{region '#Template'}
	{attribute 'Version' := '6.0.3.0'}
	{attribute 'Tags' := '"LCID": "1031", "Text": "AC, Allgemein, AHU, Startprogramm, Aggregat, Kommandierung"'}
	{attribute 'Tags' := '"LCID": "1033", "Text": "AC, General, AHU, Start program, Aggregate, Command"'}
	{attribute 'Using' := '"Type": "Template", "URI": "E_BA_AC_PlantStep01"'}
	{attribute 'Using' := '"Type": "Template", "URI": "E_BA_AC_OpMod01"'}
	{attribute 'Using' := '"Type": "Template", "URI": "Priority"'}
	{attribute 'Description' := '"LCID": "1031", "Text": "Kommandierung der Anlage FB_BA_AHU_1st_10"'}
	{attribute 'Description' := '"LCID": "1033", "Text": "Commanding the plant FB_BA_AHU_1st_10"'}
{endregion}

FUNCTION_BLOCK FB_BA_AC_PlantCmd_AHU_1st_10 EXTENDS FB_BA_View
VAR_INPUT
	eOpMode						: E_BA_AC_OpMod01;
END_VAR
VAR_OUTPUT
	ePltStp						: E_BA_AC_PlantStep01;	//	Stufen des Anlagenstarts	//	Stages of the plant starts	
	bStepCtrlUp					: BOOL;
	bStepCtrlDown				: BOOL;	
END_VAR
VAR_IN_OUT
	arrAggregate				: ARRAY [1..MAX(1,BA_Param.nMaxAggregate)] OF ST_BA_Aggregate;
END_VAR
VAR_INPUT CONSTANT
	DmpDlyCls					: FB_BA_AV_Op;
	SuAFanDlyOn					: FB_BA_AV_Op;
	ExtAFanDlyOn				: FB_BA_AV_Op;
	TempCtrlDlyOn				: FB_BA_AV_Op;
	PltStp						: FB_BA_MV_Op;
	PlantControl				: FB_BA_PlantControl;
END_VAR
VAR_INPUT CONSTANT PERSISTENT
	bInit						: BOOL := TRUE;
END_VAR
VAR
	MMuxStart					: FB_BA_MMUX_B16;
	MMuxProfile					: FB_BA_MMUX_UDI16;
	MMuxPltStp					: FB_BA_MMUX_UDI16;	//	Stufen des Anlagenstarts	//	Stages of the plant starts	
	rtrigInit					: R_TRIG;
END_VAR

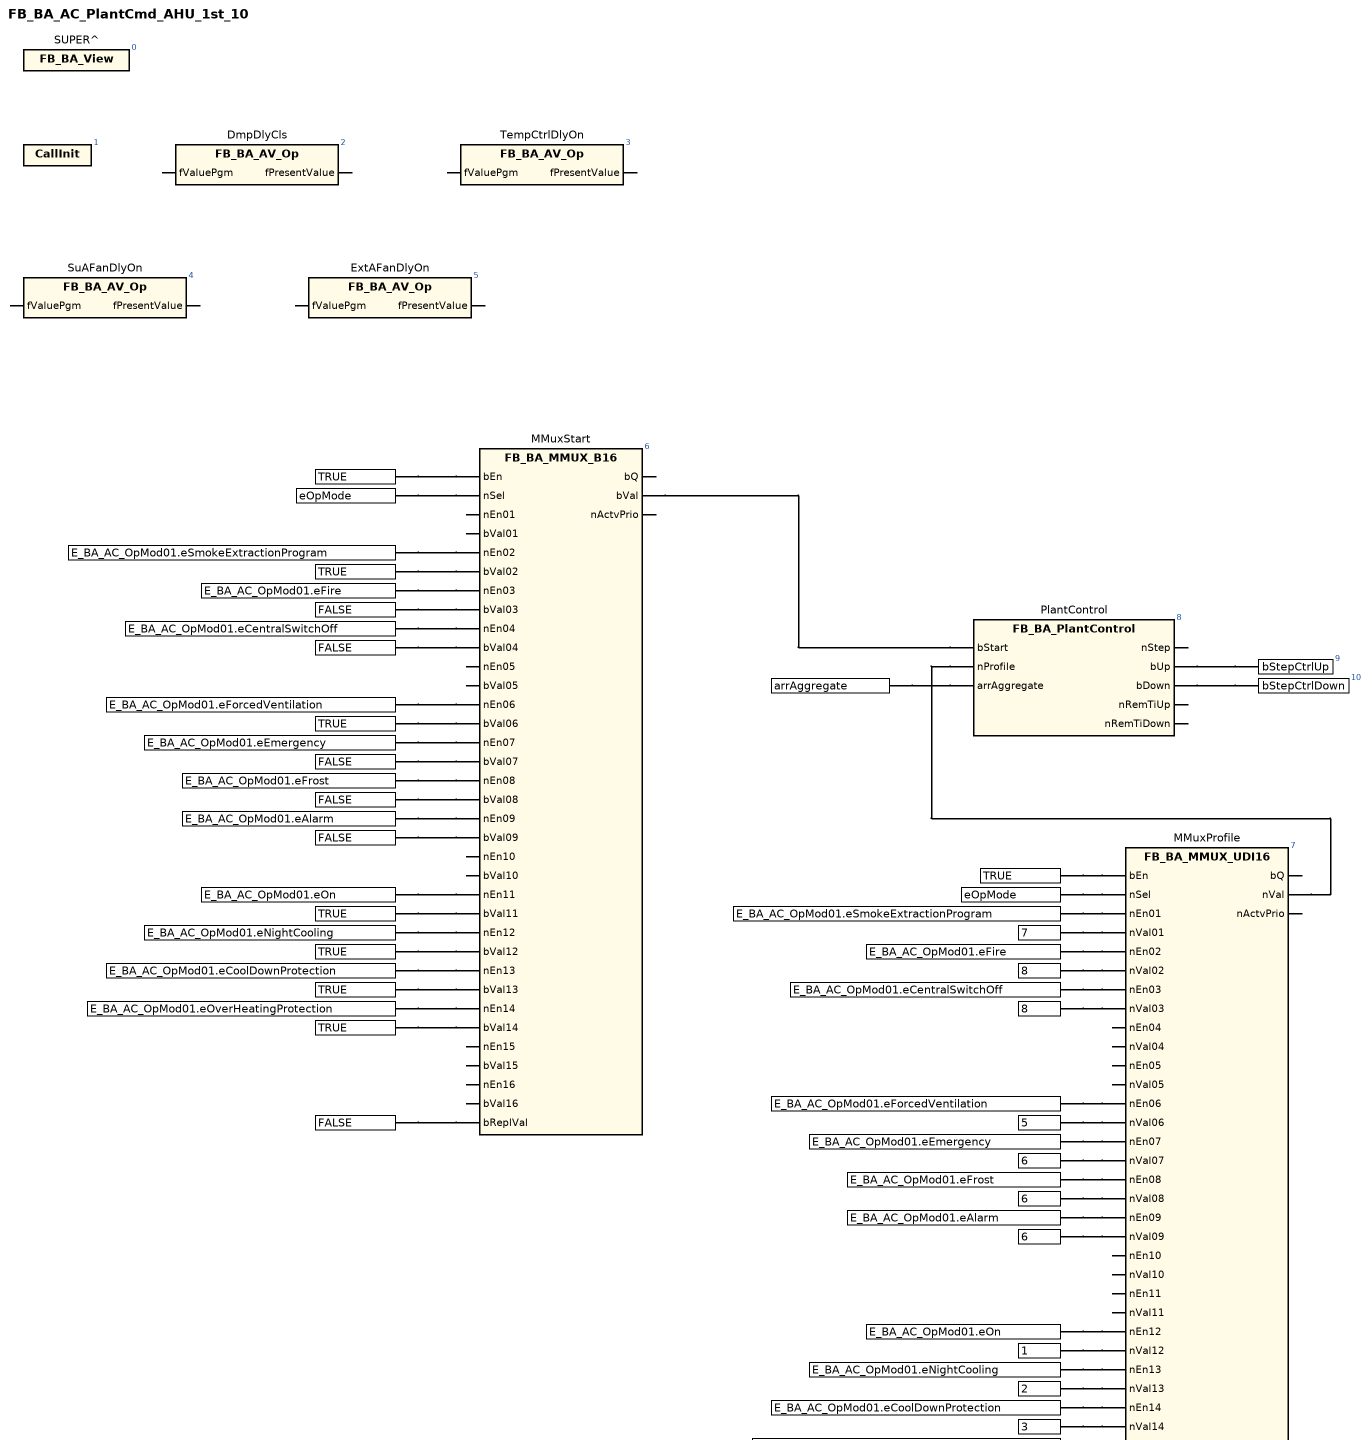
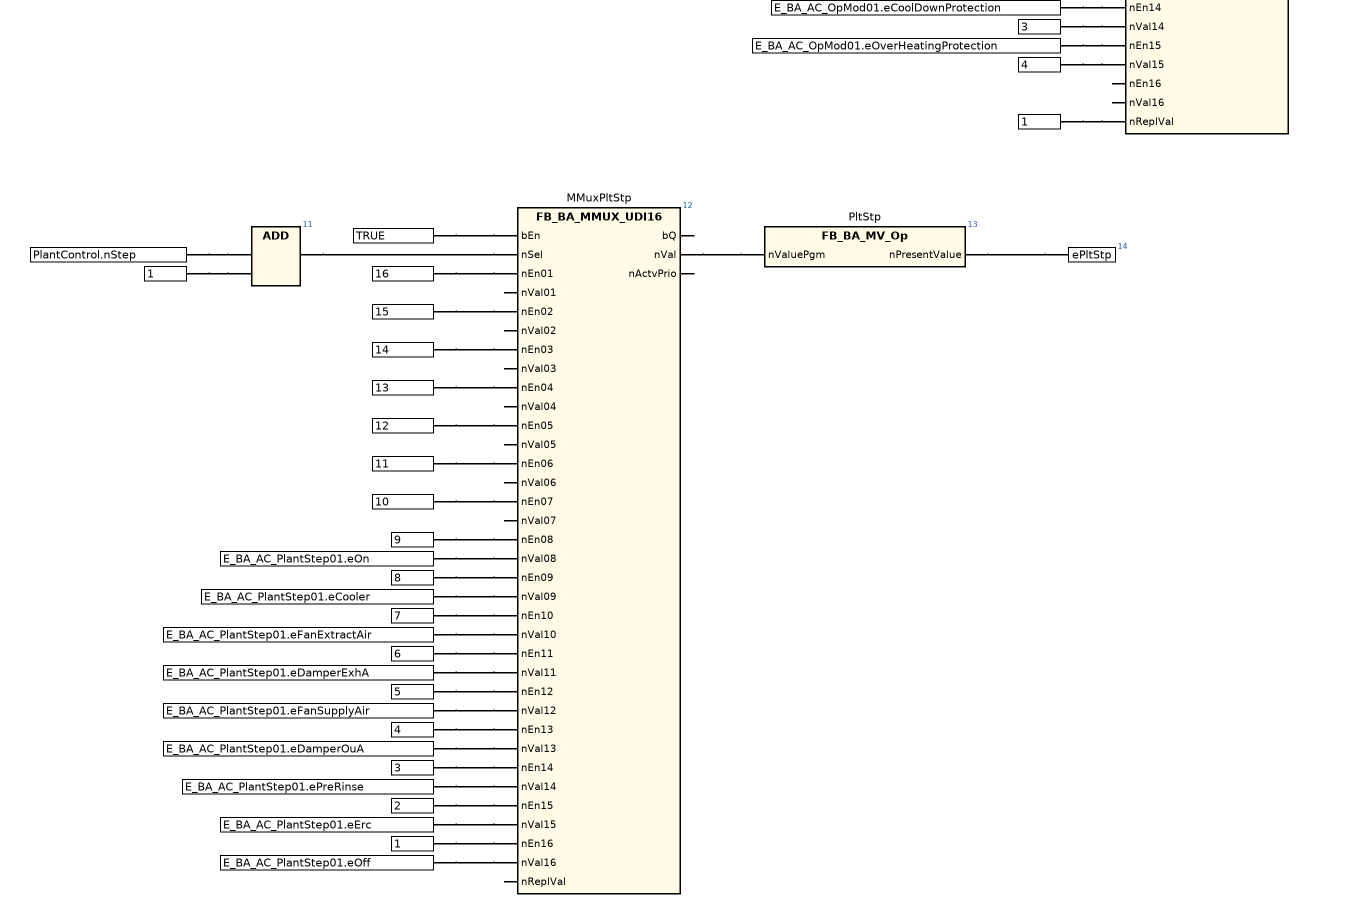
SUPER^(); // FB_BA_View
CallInit();
DmpDlyCls(); // FB_BA_AV_Op
TempCtrlDlyOn(); // FB_BA_AV_Op
SuAFanDlyOn(); // FB_BA_AV_Op
ExtAFanDlyOn(); // FB_BA_AV_Op
MMuxStart(
    bEn := TRUE,
    nSel := eOpMode,
    nEn02 := E_BA_AC_OpMod01.eSmokeExtractionProgram,
    bVal02 := TRUE,
    nEn03 := E_BA_AC_OpMod01.eFire,
    bVal03 := FALSE,
    nEn04 := E_BA_AC_OpMod01.eCentralSwitchOff,
    bVal04 := FALSE,
    nEn06 := E_BA_AC_OpMod01.eForcedVentilation,
    bVal06 := TRUE,
    nEn07 := E_BA_AC_OpMod01.eEmergency,
    bVal07 := FALSE,
    nEn08 := E_BA_AC_OpMod01.eFrost,
    bVal08 := FALSE,
    nEn09 := E_BA_AC_OpMod01.eAlarm,
    bVal09 := FALSE,
    nEn11 := E_BA_AC_OpMod01.eOn,
    bVal11 := TRUE,
    nEn12 := E_BA_AC_OpMod01.eNightCooling,
    bVal12 := TRUE,
    nEn13 := E_BA_AC_OpMod01.eCoolDownProtection,
    bVal13 := TRUE,
    nEn14 := E_BA_AC_OpMod01.eOverHeatingProtection,
    bVal14 := TRUE,
    bReplVal := FALSE); // FB_BA_MMUX_B16
MMuxProfile(
    bEn := TRUE,
    nSel := eOpMode,
    nEn01 := E_BA_AC_OpMod01.eSmokeExtractionProgram,
    nVal01 := 7,
    nEn02 := E_BA_AC_OpMod01.eFire,
    nVal02 := 8,
    nEn03 := E_BA_AC_OpMod01.eCentralSwitchOff,
    nVal03 := 8,
    nEn06 := E_BA_AC_OpMod01.eForcedVentilation,
    nVal06 := 5,
    nEn07 := E_BA_AC_OpMod01.eEmergency,
    nVal07 := 6,
    nEn08 := E_BA_AC_OpMod01.eFrost,
    nVal08 := 6,
    nEn09 := E_BA_AC_OpMod01.eAlarm,
    nVal09 := 6,
    nEn12 := E_BA_AC_OpMod01.eOn,
    nVal12 := 1,
    nEn13 := E_BA_AC_OpMod01.eNightCooling,
    nVal13 := 2,
    nEn14 := E_BA_AC_OpMod01.eCoolDownProtection,
    nVal14 := 3,
    nEn15 := E_BA_AC_OpMod01.eOverHeatingProtection,
    nVal15 := 4,
    nReplVal := 1); // FB_BA_MMUX_UDI16
PlantControl(bStart := MMuxStart.bVal, nProfile := MMuxProfile.nVal, arrAggregate := arrAggregate); // FB_BA_PlantControl
bStepCtrlUp := PlantControl.bUp;
bStepCtrlDown := PlantControl.bDown;
MMuxPltStp(
    bEn := TRUE,
    nSel := PlantControl.nStep + 1,
    nEn01 := 16,
    nEn02 := 15,
    nEn03 := 14,
    nEn04 := 13,
    nEn05 := 12,
    nEn06 := 11,
    nEn07 := 10,
    nEn08 := 9,
    nVal08 := E_BA_AC_PlantStep01.eOn,
    nEn09 := 8,
    nVal09 := E_BA_AC_PlantStep01.eCooler,
    nEn10 := 7,
    nVal10 := E_BA_AC_PlantStep01.eFanExtractAir,
    nEn11 := 6,
    nVal11 := E_BA_AC_PlantStep01.eDamperExhA,
    nEn12 := 5,
    nVal12 := E_BA_AC_PlantStep01.eFanSupplyAir,
    nEn13 := 4,
    nVal13 := E_BA_AC_PlantStep01.eDamperOuA,
    nEn14 := 3,
    nVal14 := E_BA_AC_PlantStep01.ePreRinse,
    nEn15 := 2,
    nVal15 := E_BA_AC_PlantStep01.eErc,
    nEn16 := 1,
    nVal16 := E_BA_AC_PlantStep01.eOff); // FB_BA_MMUX_UDI16
PltStp(nValuePgm := MMuxPltStp.nVal); // FB_BA_MV_Op
ePltStp := PltStp.nPresentValue;

METHOD CallInit
VAR_INPUT
END_VAR
rtrigInit.CLK := bInit;
rtrigInit();

IF	rtrigInit.Q
THEN
	ProfileDescription();

	ProfileParameter01();
	ProfileParameter02();
	ProfileParameter03();
	ProfileParameter04();
	ProfileParameter05();
	ProfileParameter06();
	ProfileParameter07();
	ProfileParameter08();
	
	StepDescription();
	
	bInit := FALSE;	
END_IF
END_METHOD

METHOD FB_init : BOOL
VAR_INPUT
	bInitRetains : BOOL; // if TRUE, the retain variables are initialized (warm start / cold start)
	bInCopyCode : BOOL;  // if TRUE, the instance afterwards gets moved into the copy code (online change)
END_VAR
DmpDlyCls.iParent			:= THIS^;
DmpDlyCls.iLabel			:= LblCtl_TimeDelayDampersClose; 	
DmpDlyCls.eUnit				:= E_BA_Unit.eTime_Seconds;  
DmpDlyCls.fValueRm			:= 15;

SuAFanDlyOn.iParent			:= THIS^;
SuAFanDlyOn.iLabel			:= LblCtl_TimeDelaySupplyAirFanOn;   		
SuAFanDlyOn.eUnit			:= E_BA_Unit.eTime_Seconds;  
SuAFanDlyOn.fValueRm		:= 10;

ExtAFanDlyOn.iParent		:= THIS^;
ExtAFanDlyOn.iLabel			:= LblCtl_TimeDelayExtractAirFanOn;   	
ExtAFanDlyOn.eUnit			:= E_BA_Unit.eTime_Seconds;  
ExtAFanDlyOn.fValueRm		:= 10;

TempCtrlDlyOn.iParent		:= THIS^;
TempCtrlDlyOn.iLabel		:= LblCtl_TimeDelayTemperatureSequenceControlOn;   	
TempCtrlDlyOn.eUnit			:= E_BA_Unit.eTime_Seconds;  
TempCtrlDlyOn.fValueRm		:= 5;

PltStp.iParent				:= THIS^;
PltStp.iLabel				:= LblCtl_StagesOfThePlantStartup; 	
PltStp.aStateText[1]		:= txtEvent_Off;
PltStp.aStateText[2]		:= txtEvent_EnergyRecovery;
PltStp.aStateText[3]		:= txtEvent_PreRinse;// or txtEvent_Preheater
PltStp.aStateText[4]		:= txtEvent_DamperOutsideAir;
PltStp.aStateText[5]		:= txtEvent_SupplyAirFan;
PltStp.aStateText[6]		:= txtEvent_DamperExhaustAir;
PltStp.aStateText[7]		:= txtEvent_ExtractAirFan;
PltStp.aStateText[8]		:= txtEvent_Cooler;
PltStp.aStateText[9]		:= txtEvent_Reheater;
PltStp.aStateText[10]		:= txtEvent_MixedAir;
PltStp.aStateText[11]		:= txtEvent_EnableTemperatureControl;
PltStp.aStateText[12]		:= txtEvent_EnableHumidityControl;
PltStp.aStateText[13]		:= txtEvent_On;
END_METHOD

METHOD ProfileDescription
VAR
END_VAR
PlantControl.arrProfileDescription[1].sDescription	:= txtEvent_Auto;		
PlantControl.arrProfileDescription[1].nPrio			:= Priority.nProgram;

PlantControl.arrProfileDescription[2].sDescription	:= txtEvent_NightCooling;
PlantControl.arrProfileDescription[2].nPrio			:= Priority.nProgram;

PlantControl.arrProfileDescription[3].sDescription	:= txtEvent_CoolDownProtection; 		
PlantControl.arrProfileDescription[3].nPrio			:= Priority.nProgram;

PlantControl.arrProfileDescription[4].sDescription	:= txtEvent_OverHeatingProtection;
PlantControl.arrProfileDescription[4].nPrio			:= Priority.nProgram;

PlantControl.arrProfileDescription[5].sDescription	:= txtEvent_ForcedVentilation;
PlantControl.arrProfileDescription[5].nPrio			:= Priority.nCritical;

PlantControl.arrProfileDescription[6].sDescription	:= txtEvent_CriticalOff;
PlantControl.arrProfileDescription[6].nPrio			:= Priority.nCritical;

PlantControl.arrProfileDescription[7].sDescription	:= txtEvent_SmokeExtraction_P;
PlantControl.arrProfileDescription[7].nPrio			:= Priority.nLifeSafety;

PlantControl.arrProfileDescription[8].sDescription	:= txtEvent_LifeSafetyOff;
PlantControl.arrProfileDescription[8].nPrio			:= Priority.nLifeSafety;
END_METHOD

METHOD ProfileParameter01
VAR
END_VAR
// Profile Auto
// PlantControl.arrProfileParameter[Profile,Step]
// Step 1 = Erc, 
// Step 2 = PreHtr
// Step 3 = DamperOuA
// Step 4 = FanSupplyAir
// Step 5 = DamperExhA
// Step 6 = FanExtractAir
// Step 7 = Cooler
// Step 8 = EnablingTemperatureControl

PlantControl.arrProfileParameter[1,1].bValue			:= TRUE;		
PlantControl.arrProfileParameter[1,1].nValue			:= 0;
PlantControl.arrProfileParameter[1,1].fValue			:= 0;		
PlantControl.arrProfileParameter[1,1].fDelayUp			:= 0;	
PlantControl.arrProfileParameter[1,1].fDelayDown		:= 0;	
PlantControl.arrProfileParameter[1,1].bEnFdbUp			:= FALSE;	
PlantControl.arrProfileParameter[1,1].bEnFdbDown		:= FALSE;	
                          
PlantControl.arrProfileParameter[1,2].bValue			:= TRUE;		
PlantControl.arrProfileParameter[1,2].nValue			:= 0;		
PlantControl.arrProfileParameter[1,2].fValue			:= 0;		
PlantControl.arrProfileParameter[1,2].fDelayUp			:= 0;	
PlantControl.arrProfileParameter[1,2].fDelayDown		:= 0;	
PlantControl.arrProfileParameter[1,2].bEnFdbUp			:= TRUE;	
PlantControl.arrProfileParameter[1,2].bEnFdbDown		:= FALSE;	
                          
PlantControl.arrProfileParameter[1,3].bValue			:= TRUE;		
PlantControl.arrProfileParameter[1,3].nValue			:= 0;		
PlantControl.arrProfileParameter[1,3].fValue			:= 0;		
PlantControl.arrProfileParameter[1,3].fDelayUp			:= SuAFanDlyOn.fPresentValue;	
PlantControl.arrProfileParameter[1,3].fDelayDown		:= 0;	
PlantControl.arrProfileParameter[1,3].bEnFdbUp			:= TRUE;	
PlantControl.arrProfileParameter[1,3].bEnFdbDown		:= FALSE;	
                          
PlantControl.arrProfileParameter[1,4].bValue			:= FALSE;		
PlantControl.arrProfileParameter[1,4].nValue			:= E_BA_Mdlt.eOn;		
PlantControl.arrProfileParameter[1,4].fValue			:= 0;		
PlantControl.arrProfileParameter[1,4].fDelayUp			:= 0;	
PlantControl.arrProfileParameter[1,4].fDelayDown		:= DmpDlyCls.fPresentValue;	
PlantControl.arrProfileParameter[1,4].bEnFdbUp			:= FALSE;	
PlantControl.arrProfileParameter[1,4].bEnFdbDown		:= FALSE;	
                          
PlantControl.arrProfileParameter[1,5].bValue			:= TRUE;		
PlantControl.arrProfileParameter[1,5].nValue			:= 0;		
PlantControl.arrProfileParameter[1,5].fValue			:= 0;		
PlantControl.arrProfileParameter[1,5].fDelayUp			:= ExtAFanDlyOn.fPresentValue;	
PlantControl.arrProfileParameter[1,5].fDelayDown		:= 0;	
PlantControl.arrProfileParameter[1,5].bEnFdbUp			:= TRUE;	
PlantControl.arrProfileParameter[1,5].bEnFdbDown		:= FALSE;	
                          
PlantControl.arrProfileParameter[1,6].bValue			:= FALSE;		
PlantControl.arrProfileParameter[1,6].nValue			:= E_BA_Mdlt.eOn;		
PlantControl.arrProfileParameter[1,6].fValue			:= 0;		
PlantControl.arrProfileParameter[1,6].fDelayUp			:= 0;	
PlantControl.arrProfileParameter[1,6].fDelayDown		:= DmpDlyCls.fPresentValue;	
PlantControl.arrProfileParameter[1,6].bEnFdbUp			:= FALSE;	
PlantControl.arrProfileParameter[1,6].bEnFdbDown		:= FALSE;	
                          
PlantControl.arrProfileParameter[1,7].bValue			:= TRUE;		
PlantControl.arrProfileParameter[1,7].nValue			:= 0;		
PlantControl.arrProfileParameter[1,7].fValue			:= 0;		
PlantControl.arrProfileParameter[1,7].fDelayUp			:= TempCtrlDlyOn.fPresentValue;	
PlantControl.arrProfileParameter[1,7].fDelayDown		:= 0;	
PlantControl.arrProfileParameter[1,7].bEnFdbUp			:= FALSE;	
PlantControl.arrProfileParameter[1,7].bEnFdbDown		:= FALSE;	
                          
PlantControl.arrProfileParameter[1,8].bValue			:= FALSE;		
PlantControl.arrProfileParameter[1,8].nValue			:= E_BA_Mdlt.eOn;		
PlantControl.arrProfileParameter[1,8].fValue			:= 0;		
PlantControl.arrProfileParameter[1,8].fDelayUp			:= 0;	
PlantControl.arrProfileParameter[1,8].fDelayDown		:= 0;	
PlantControl.arrProfileParameter[1,8].bEnFdbUp			:= FALSE;	
PlantControl.arrProfileParameter[1,8].bEnFdbDown		:= FALSE;
END_METHOD

METHOD ProfileParameter02
VAR
END_VAR
// Profile NightCooling
// PlantControl.arrProfileParameter[Profile,Step]
// Step 1 = Erc, 
// Step 2 = PreHtr
// Step 3 = DamperOuA
// Step 4 = FanSupplyAir
// Step 5 = DamperExhA
// Step 6 = FanExtractAir
// Step 7 = Cooler
// Step 8 = EnablingTemperatureControl

PlantControl.arrProfileParameter[2,1].bValue			:= FALSE;		
PlantControl.arrProfileParameter[2,1].nValue			:= 0;
PlantControl.arrProfileParameter[2,1].fValue			:= 0;		
PlantControl.arrProfileParameter[2,1].fDelayUp			:= 0;	
PlantControl.arrProfileParameter[2,1].fDelayDown		:= 0;	
PlantControl.arrProfileParameter[2,1].bEnFdbUp			:= FALSE;	
PlantControl.arrProfileParameter[2,1].bEnFdbDown		:= FALSE;	
                          
PlantControl.arrProfileParameter[2,2].bValue			:= FALSE;		
PlantControl.arrProfileParameter[2,2].nValue			:= 0;		
PlantControl.arrProfileParameter[2,2].fValue			:= 0;		
PlantControl.arrProfileParameter[2,2].fDelayUp			:= 0;	
PlantControl.arrProfileParameter[2,2].fDelayDown		:= 0;	
PlantControl.arrProfileParameter[2,2].bEnFdbUp			:= FALSE;	
PlantControl.arrProfileParameter[2,2].bEnFdbDown		:= FALSE;	
                          
PlantControl.arrProfileParameter[2,3].bValue			:= TRUE;		
PlantControl.arrProfileParameter[2,3].nValue			:= 0;		
PlantControl.arrProfileParameter[2,3].fValue			:= 0;		
PlantControl.arrProfileParameter[2,3].fDelayUp			:= SuAFanDlyOn.fPresentValue;	
PlantControl.arrProfileParameter[2,3].fDelayDown		:= 0;	
PlantControl.arrProfileParameter[2,3].bEnFdbUp			:= TRUE;	
PlantControl.arrProfileParameter[2,3].bEnFdbDown		:= FALSE;	
                          
PlantControl.arrProfileParameter[2,4].bValue			:= FALSE;		
PlantControl.arrProfileParameter[2,4].nValue			:= E_BA_Mdlt.eMax;		
PlantControl.arrProfileParameter[2,4].fValue			:= 0;		
PlantControl.arrProfileParameter[2,4].fDelayUp			:= 0;	
PlantControl.arrProfileParameter[2,4].fDelayDown		:= 0;	
PlantControl.arrProfileParameter[2,4].bEnFdbUp			:= FALSE;	
PlantControl.arrProfileParameter[2,4].bEnFdbDown		:= FALSE;	
                          
PlantControl.arrProfileParameter[2,5].bValue			:= TRUE;		
PlantControl.arrProfileParameter[2,5].nValue			:= 0;		
PlantControl.arrProfileParameter[2,5].fValue			:= 0;		
PlantControl.arrProfileParameter[2,5].fDelayUp			:= ExtAFanDlyOn.fPresentValue;	
PlantControl.arrProfileParameter[2,5].fDelayDown		:= 0;	
PlantControl.arrProfileParameter[2,5].bEnFdbUp			:= TRUE;	
PlantControl.arrProfileParameter[2,5].bEnFdbDown		:= FALSE;	
                          
PlantControl.arrProfileParameter[2,6].bValue			:= FALSE;		
PlantControl.arrProfileParameter[2,6].nValue			:= E_BA_Mdlt.eMax;		
PlantControl.arrProfileParameter[2,6].fValue			:= 0;		
PlantControl.arrProfileParameter[2,6].fDelayUp			:= 0;	
PlantControl.arrProfileParameter[2,6].fDelayDown		:= 0;	
PlantControl.arrProfileParameter[2,6].bEnFdbUp			:= FALSE;	
PlantControl.arrProfileParameter[2,6].bEnFdbDown		:= FALSE;	
                          
PlantControl.arrProfileParameter[2,7].bValue			:= FALSE;		
PlantControl.arrProfileParameter[2,7].nValue			:= 0;		
PlantControl.arrProfileParameter[2,7].fValue			:= 0;		
PlantControl.arrProfileParameter[2,7].fDelayUp			:= 0;	
PlantControl.arrProfileParameter[2,7].fDelayDown		:= 0;	
PlantControl.arrProfileParameter[2,7].bEnFdbUp			:= FALSE;	
PlantControl.arrProfileParameter[2,7].bEnFdbDown		:= FALSE;	
                          
PlantControl.arrProfileParameter[2,8].bValue			:= FALSE;		
PlantControl.arrProfileParameter[2,8].nValue			:= E_BA_Mdlt.eOff;		
PlantControl.arrProfileParameter[2,8].fValue			:= 0;		
PlantControl.arrProfileParameter[2,8].fDelayUp			:= 0;	
PlantControl.arrProfileParameter[2,8].fDelayDown		:= 0;	
PlantControl.arrProfileParameter[2,8].bEnFdbUp			:= FALSE;	
PlantControl.arrProfileParameter[2,8].bEnFdbDown		:= FALSE;
END_METHOD

METHOD ProfileParameter03
VAR
END_VAR
// Profile CoolDownProtection
// PlantControl.arrProfileParameter[Profile,Step]
// Step 1 = Erc, 
// Step 2 = PreHtr
// Step 3 = DamperOuA
// Step 4 = FanSupplyAir
// Step 5 = DamperExhA
// Step 6 = FanExtractAir
// Step 7 = Cooler
// Step 8 = EnablingTemperatureControl

PlantControl.arrProfileParameter[3,1].bValue			:= TRUE;		
PlantControl.arrProfileParameter[3,1].nValue			:= 0;
PlantControl.arrProfileParameter[3,1].fValue			:= 0;		
PlantControl.arrProfileParameter[3,1].fDelayUp			:= 0;	
PlantControl.arrProfileParameter[3,1].fDelayDown		:= 0;	
PlantControl.arrProfileParameter[3,1].bEnFdbUp			:= FALSE;	
PlantControl.arrProfileParameter[3,1].bEnFdbDown		:= FALSE;	
                          
PlantControl.arrProfileParameter[3,2].bValue			:= TRUE;		
PlantControl.arrProfileParameter[3,2].nValue			:= 0;		
PlantControl.arrProfileParameter[3,2].fValue			:= 0;		
PlantControl.arrProfileParameter[3,2].fDelayUp			:= 0;	
PlantControl.arrProfileParameter[3,2].fDelayDown		:= 0;	
PlantControl.arrProfileParameter[3,2].bEnFdbUp			:= TRUE;	
PlantControl.arrProfileParameter[3,2].bEnFdbDown		:= FALSE;	
                          
PlantControl.arrProfileParameter[3,3].bValue			:= TRUE;		
PlantControl.arrProfileParameter[3,3].nValue			:= 0;		
PlantControl.arrProfileParameter[3,3].fValue			:= 0;		
PlantControl.arrProfileParameter[3,3].fDelayUp			:= SuAFanDlyOn.fPresentValue;	
PlantControl.arrProfileParameter[3,3].fDelayDown		:= 0;	
PlantControl.arrProfileParameter[3,3].bEnFdbUp			:= TRUE;	
PlantControl.arrProfileParameter[3,3].bEnFdbDown		:= FALSE;	
                          
PlantControl.arrProfileParameter[3,4].bValue			:= FALSE;		
PlantControl.arrProfileParameter[3,4].nValue			:= E_BA_Mdlt.eMax;		
PlantControl.arrProfileParameter[3,4].fValue			:= 0;		
PlantControl.arrProfileParameter[3,4].fDelayUp			:= 0;	
PlantControl.arrProfileParameter[3,4].fDelayDown		:= 0;	
PlantControl.arrProfileParameter[3,4].bEnFdbUp			:= FALSE;	
PlantControl.arrProfileParameter[3,4].bEnFdbDown		:= FALSE;	
                          
PlantControl.arrProfileParameter[3,5].bValue			:= TRUE;		
PlantControl.arrProfileParameter[3,5].nValue			:= 0;		
PlantControl.arrProfileParameter[3,5].fValue			:= 0;		
PlantControl.arrProfileParameter[3,5].fDelayUp			:= ExtAFanDlyOn.fPresentValue;	
PlantControl.arrProfileParameter[3,5].fDelayDown		:= 0;	
PlantControl.arrProfileParameter[3,5].bEnFdbUp			:= TRUE;	
PlantControl.arrProfileParameter[3,5].bEnFdbDown		:= FALSE;	
                          
PlantControl.arrProfileParameter[3,6].bValue			:= FALSE;		
PlantControl.arrProfileParameter[3,6].nValue			:= E_BA_Mdlt.eMax;		
PlantControl.arrProfileParameter[3,6].fValue			:= 0;		
PlantControl.arrProfileParameter[3,6].fDelayUp			:= 0;	
PlantControl.arrProfileParameter[3,6].fDelayDown		:= 0;	
PlantControl.arrProfileParameter[3,6].bEnFdbUp			:= FALSE;	
PlantControl.arrProfileParameter[3,6].bEnFdbDown		:= FALSE;	
                          
PlantControl.arrProfileParameter[3,7].bValue			:= FALSE;		
PlantControl.arrProfileParameter[3,7].nValue			:= 0;		
PlantControl.arrProfileParameter[3,7].fValue			:= 0;		
PlantControl.arrProfileParameter[3,7].fDelayUp			:= 0;	
PlantControl.arrProfileParameter[3,7].fDelayDown		:= 0;	
PlantControl.arrProfileParameter[3,7].bEnFdbUp			:= FALSE;	
PlantControl.arrProfileParameter[3,7].bEnFdbDown		:= FALSE;	
                          
PlantControl.arrProfileParameter[3,8].bValue			:= FALSE;		
PlantControl.arrProfileParameter[3,8].nValue			:= E_BA_Mdlt.eMax;		
PlantControl.arrProfileParameter[3,8].fValue			:= 0;		
PlantControl.arrProfileParameter[3,8].fDelayUp			:= 0;	
PlantControl.arrProfileParameter[3,8].fDelayDown		:= 0;	
PlantControl.arrProfileParameter[3,8].bEnFdbUp			:= FALSE;	
PlantControl.arrProfileParameter[3,8].bEnFdbDown		:= FALSE;
END_METHOD

METHOD ProfileParameter04
VAR
END_VAR
// Profile OverHeatingProtection
// PlantControl.arrProfileParameter[Profile,Step]
// Step 1 = Erc, 
// Step 2 = PreHtr
// Step 3 = DamperOuA
// Step 4 = FanSupplyAir
// Step 5 = DamperExhA
// Step 6 = FanExtractAir
// Step 7 = Cooler
// Step 8 = EnablingTemperatureControl

PlantControl.arrProfileParameter[4,1].bValue			:= TRUE;		
PlantControl.arrProfileParameter[4,1].nValue			:= 0;
PlantControl.arrProfileParameter[4,1].fValue			:= 0;		
PlantControl.arrProfileParameter[4,1].fDelayUp			:= 0;	
PlantControl.arrProfileParameter[4,1].fDelayDown		:= 0;	
PlantControl.arrProfileParameter[4,1].bEnFdbUp			:= FALSE;	
PlantControl.arrProfileParameter[4,1].bEnFdbDown		:= FALSE;	
                          
PlantControl.arrProfileParameter[4,2].bValue			:= FALSE;		
PlantControl.arrProfileParameter[4,2].nValue			:= 0;		
PlantControl.arrProfileParameter[4,2].fValue			:= 0;		
PlantControl.arrProfileParameter[4,2].fDelayUp			:= 0;	
PlantControl.arrProfileParameter[4,2].fDelayDown		:= 0;	
PlantControl.arrProfileParameter[4,2].bEnFdbUp			:= FALSE;	
PlantControl.arrProfileParameter[4,2].bEnFdbDown		:= FALSE;	
                          
PlantControl.arrProfileParameter[4,3].bValue			:= TRUE;		
PlantControl.arrProfileParameter[4,3].nValue			:= 0;		
PlantControl.arrProfileParameter[4,3].fValue			:= 0;		
PlantControl.arrProfileParameter[4,3].fDelayUp			:= SuAFanDlyOn.fPresentValue;	
PlantControl.arrProfileParameter[4,3].fDelayDown		:= 0;	
PlantControl.arrProfileParameter[4,3].bEnFdbUp			:= TRUE;	
PlantControl.arrProfileParameter[4,3].bEnFdbDown		:= FALSE;	
                          
PlantControl.arrProfileParameter[4,4].bValue			:= FALSE;		
PlantControl.arrProfileParameter[4,4].nValue			:= E_BA_Mdlt.eOn;		
PlantControl.arrProfileParameter[4,4].fValue			:= 0;		
PlantControl.arrProfileParameter[4,4].fDelayUp			:= 0;	
PlantControl.arrProfileParameter[4,4].fDelayDown		:= 0;	
PlantControl.arrProfileParameter[4,4].bEnFdbUp			:= FALSE;	
PlantControl.arrProfileParameter[4,4].bEnFdbDown		:= FALSE;	
                          
PlantControl.arrProfileParameter[4,5].bValue			:= TRUE;		
PlantControl.arrProfileParameter[4,5].nValue			:= 0;		
PlantControl.arrProfileParameter[4,5].fValue			:= 0;		
PlantControl.arrProfileParameter[4,5].fDelayUp			:= ExtAFanDlyOn.fPresentValue;	
PlantControl.arrProfileParameter[4,5].fDelayDown		:= 0;	
PlantControl.arrProfileParameter[4,5].bEnFdbUp			:= TRUE;	
PlantControl.arrProfileParameter[4,5].bEnFdbDown		:= FALSE;	
                          
PlantControl.arrProfileParameter[4,6].bValue			:= FALSE;		
PlantControl.arrProfileParameter[4,6].nValue			:= E_BA_Mdlt.eOn;		
PlantControl.arrProfileParameter[4,6].fValue			:= 0;		
PlantControl.arrProfileParameter[4,6].fDelayUp			:= 0;	
PlantControl.arrProfileParameter[4,6].fDelayDown		:= 0;	
PlantControl.arrProfileParameter[4,6].bEnFdbUp			:= FALSE;	
PlantControl.arrProfileParameter[4,6].bEnFdbDown		:= FALSE;	
                          
PlantControl.arrProfileParameter[4,7].bValue			:= TRUE;		
PlantControl.arrProfileParameter[4,7].nValue			:= 0;		
PlantControl.arrProfileParameter[4,7].fValue			:= 0;		
PlantControl.arrProfileParameter[4,7].fDelayUp			:= 0;	
PlantControl.arrProfileParameter[4,7].fDelayDown		:= 0;	
PlantControl.arrProfileParameter[4,7].bEnFdbUp			:= FALSE;	
PlantControl.arrProfileParameter[4,7].bEnFdbDown		:= FALSE;	
                          
PlantControl.arrProfileParameter[4,8].bValue			:= FALSE;		
PlantControl.arrProfileParameter[4,8].nValue			:= E_BA_Mdlt.eMin;		
PlantControl.arrProfileParameter[4,8].fValue			:= 0;		
PlantControl.arrProfileParameter[4,8].fDelayUp			:= 0;	
PlantControl.arrProfileParameter[4,8].fDelayDown		:= 0;	
PlantControl.arrProfileParameter[4,8].bEnFdbUp			:= FALSE;	
PlantControl.arrProfileParameter[4,8].bEnFdbDown		:= FALSE;
END_METHOD

METHOD ProfileParameter05
VAR
END_VAR
// Profile ForcedVentilation
// PlantControl.arrProfileParameter[Profile,Step]
// Step 1 = Erc, 
// Step 2 = PreHtr
// Step 3 = DamperOuA
// Step 4 = FanSupplyAir
// Step 5 = DamperExhA
// Step 6 = FanExtractAir
// Step 7 = Cooler
// Step 8 = EnablingTemperatureControl

PlantControl.arrProfileParameter[5,1].bValue			:= TRUE;		
PlantControl.arrProfileParameter[5,1].nValue			:= 0;
PlantControl.arrProfileParameter[5,1].fValue			:= 0;		
PlantControl.arrProfileParameter[5,1].fDelayUp			:= 0;	
PlantControl.arrProfileParameter[5,1].fDelayDown		:= 0;	
PlantControl.arrProfileParameter[5,1].bEnFdbUp			:= FALSE;	
PlantControl.arrProfileParameter[5,1].bEnFdbDown		:= FALSE;	
                          
PlantControl.arrProfileParameter[5,2].bValue			:= TRUE;		
PlantControl.arrProfileParameter[5,2].nValue			:= 0;		
PlantControl.arrProfileParameter[5,2].fValue			:= 0;		
PlantControl.arrProfileParameter[5,2].fDelayUp			:= 0;	
PlantControl.arrProfileParameter[5,2].fDelayDown		:= 0;	
PlantControl.arrProfileParameter[5,2].bEnFdbUp			:= FALSE;	
PlantControl.arrProfileParameter[5,2].bEnFdbDown		:= FALSE;	
                          
PlantControl.arrProfileParameter[5,3].bValue			:= TRUE;		
PlantControl.arrProfileParameter[5,3].nValue			:= 0;		
PlantControl.arrProfileParameter[5,3].fValue			:= 0;		
PlantControl.arrProfileParameter[5,3].fDelayUp			:= 0;	
PlantControl.arrProfileParameter[5,3].fDelayDown		:= 0;	
PlantControl.arrProfileParameter[5,3].bEnFdbUp			:= TRUE;	
PlantControl.arrProfileParameter[5,3].bEnFdbDown		:= FALSE;	
                          
PlantControl.arrProfileParameter[5,4].bValue			:= FALSE;		
PlantControl.arrProfileParameter[5,4].nValue			:= E_BA_Mdlt.eMax;		
PlantControl.arrProfileParameter[5,4].fValue			:= 0;		
PlantControl.arrProfileParameter[5,4].fDelayUp			:= 0;	
PlantControl.arrProfileParameter[5,4].fDelayDown		:= 0;	
PlantControl.arrProfileParameter[5,4].bEnFdbUp			:= FALSE;	
PlantControl.arrProfileParameter[5,4].bEnFdbDown		:= FALSE;	
                          
PlantControl.arrProfileParameter[5,5].bValue			:= TRUE;		
PlantControl.arrProfileParameter[5,5].nValue			:= 0;		
PlantControl.arrProfileParameter[5,5].fValue			:= 0;		
PlantControl.arrProfileParameter[5,5].fDelayUp			:= 0;	
PlantControl.arrProfileParameter[5,5].fDelayDown		:= 0;	
PlantControl.arrProfileParameter[5,5].bEnFdbUp			:= TRUE;	
PlantControl.arrProfileParameter[5,5].bEnFdbDown		:= FALSE;	
                          
PlantControl.arrProfileParameter[5,6].bValue			:= FALSE;		
PlantControl.arrProfileParameter[5,6].nValue			:= E_BA_Mdlt.eMax;		
PlantControl.arrProfileParameter[5,6].fValue			:= 0;		
PlantControl.arrProfileParameter[5,6].fDelayUp			:= 0;	
PlantControl.arrProfileParameter[5,6].fDelayDown		:= 0;	
PlantControl.arrProfileParameter[5,6].bEnFdbUp			:= FALSE;	
PlantControl.arrProfileParameter[5,6].bEnFdbDown		:= FALSE;	
                          
PlantControl.arrProfileParameter[5,7].bValue			:= TRUE;		
PlantControl.arrProfileParameter[5,7].nValue			:= 0;		
PlantControl.arrProfileParameter[5,7].fValue			:= 0;		
PlantControl.arrProfileParameter[5,7].fDelayUp			:= 0;	
PlantControl.arrProfileParameter[5,7].fDelayDown		:= 0;	
PlantControl.arrProfileParameter[5,7].bEnFdbUp			:= FALSE;	
PlantControl.arrProfileParameter[5,7].bEnFdbDown		:= FALSE;	
                          
PlantControl.arrProfileParameter[5,8].bValue			:= FALSE;		
PlantControl.arrProfileParameter[5,8].nValue			:= E_BA_Mdlt.eOn;		
PlantControl.arrProfileParameter[5,8].fValue			:= 0;		
PlantControl.arrProfileParameter[5,8].fDelayUp			:= 0;	
PlantControl.arrProfileParameter[5,8].fDelayDown		:= 0;	
PlantControl.arrProfileParameter[5,8].bEnFdbUp			:= FALSE;	
PlantControl.arrProfileParameter[5,8].bEnFdbDown		:= FALSE;
END_METHOD

METHOD ProfileParameter06
VAR
END_VAR
// Profile CriticalOff
// PlantControl.arrProfileParameter[Profile,Step]
// Step 1 = Erc, 
// Step 2 = PreHtr
// Step 3 = DamperOuA
// Step 4 = FanSupplyAir
// Step 5 = DamperExhA
// Step 6 = FanExtractAir
// Step 7 = Cooler
// Step 8 = EnablingTemperatureControl

PlantControl.arrProfileParameter[6,1].bValue			:= FALSE;		
PlantControl.arrProfileParameter[6,1].nValue			:= 0;
PlantControl.arrProfileParameter[6,1].fValue			:= 0;		
PlantControl.arrProfileParameter[6,1].fDelayUp			:= 0;	
PlantControl.arrProfileParameter[6,1].fDelayDown		:= 0;	
PlantControl.arrProfileParameter[6,1].bEnFdbUp			:= FALSE;	
PlantControl.arrProfileParameter[6,1].bEnFdbDown		:= FALSE;	
                          
PlantControl.arrProfileParameter[6,2].bValue			:= FALSE;		
PlantControl.arrProfileParameter[6,2].nValue			:= 0;		
PlantControl.arrProfileParameter[6,2].fValue			:= 0;		
PlantControl.arrProfileParameter[6,2].fDelayUp			:= 0;	
PlantControl.arrProfileParameter[6,2].fDelayDown		:= 0;	
PlantControl.arrProfileParameter[6,2].bEnFdbUp			:= FALSE;	
PlantControl.arrProfileParameter[6,2].bEnFdbDown		:= FALSE;	
                          
PlantControl.arrProfileParameter[6,3].bValue			:= FALSE;		
PlantControl.arrProfileParameter[6,3].nValue			:= 0;		
PlantControl.arrProfileParameter[6,3].fValue			:= 0;		
PlantControl.arrProfileParameter[6,3].fDelayUp			:= 0;	
PlantControl.arrProfileParameter[6,3].fDelayDown		:= 0;	
PlantControl.arrProfileParameter[6,3].bEnFdbUp			:= FALSE;	
PlantControl.arrProfileParameter[6,3].bEnFdbDown		:= FALSE;	
                          
PlantControl.arrProfileParameter[6,4].bValue			:= FALSE;		
PlantControl.arrProfileParameter[6,4].nValue			:= E_BA_Mdlt.eOff;		
PlantControl.arrProfileParameter[6,4].fValue			:= 0;		
PlantControl.arrProfileParameter[6,4].fDelayUp			:= 0;	
PlantControl.arrProfileParameter[6,4].fDelayDown		:= 0;	
PlantControl.arrProfileParameter[6,4].bEnFdbUp			:= FALSE;	
PlantControl.arrProfileParameter[6,4].bEnFdbDown		:= FALSE;	
                          
PlantControl.arrProfileParameter[6,5].bValue			:= FALSE;		
PlantControl.arrProfileParameter[6,5].nValue			:= 0;		
PlantControl.arrProfileParameter[6,5].fValue			:= 0;		
PlantControl.arrProfileParameter[6,5].fDelayUp			:= 0;	
PlantControl.arrProfileParameter[6,5].fDelayDown		:= 0;	
PlantControl.arrProfileParameter[6,5].bEnFdbUp			:= FALSE;	
PlantControl.arrProfileParameter[6,5].bEnFdbDown		:= FALSE;	
                          
PlantControl.arrProfileParameter[6,6].bValue			:= FALSE;		
PlantControl.arrProfileParameter[6,6].nValue			:= E_BA_Mdlt.eOff;		
PlantControl.arrProfileParameter[6,6].fValue			:= 0;		
PlantControl.arrProfileParameter[6,6].fDelayUp			:= 0;	
PlantControl.arrProfileParameter[6,6].fDelayDown		:= 0;	
PlantControl.arrProfileParameter[6,6].bEnFdbUp			:= FALSE;	
PlantControl.arrProfileParameter[6,6].bEnFdbDown		:= FALSE;	
                          
PlantControl.arrProfileParameter[6,7].bValue			:= FALSE;		
PlantControl.arrProfileParameter[6,7].nValue			:= 0;		
PlantControl.arrProfileParameter[6,7].fValue			:= 0;		
PlantControl.arrProfileParameter[6,7].fDelayUp			:= 0;	
PlantControl.arrProfileParameter[6,7].fDelayDown		:= 0;	
PlantControl.arrProfileParameter[6,7].bEnFdbUp			:= FALSE;	
PlantControl.arrProfileParameter[6,7].bEnFdbDown		:= FALSE;	
                          
PlantControl.arrProfileParameter[6,8].bValue			:= FALSE;		
PlantControl.arrProfileParameter[6,8].nValue			:= E_BA_Mdlt.eOff;		
PlantControl.arrProfileParameter[6,8].fValue			:= 0;		
PlantControl.arrProfileParameter[6,8].fDelayUp			:= 0;	
PlantControl.arrProfileParameter[6,8].fDelayDown		:= 0;	
PlantControl.arrProfileParameter[6,8].bEnFdbUp			:= FALSE;	
PlantControl.arrProfileParameter[6,8].bEnFdbDown		:= FALSE;
END_METHOD

METHOD ProfileParameter07
VAR
END_VAR
// Profile SmokeExtractionProgram
// PlantControl.arrProfileParameter[Profile,Step]
// Step 1 = Erc, 
// Step 2 = PreHtr
// Step 3 = DamperOuA
// Step 4 = FanSupplyAir
// Step 5 = DamperExhA
// Step 6 = FanExtractAir
// Step 7 = Cooler
// Step 8 = EnablingTemperatureControl

PlantControl.arrProfileParameter[7,1].bValue			:= FALSE;		
PlantControl.arrProfileParameter[7,1].nValue			:= 0;
PlantControl.arrProfileParameter[7,1].fValue			:= 0;		
PlantControl.arrProfileParameter[7,1].fDelayUp			:= 0;	
PlantControl.arrProfileParameter[7,1].fDelayDown		:= 0;	
PlantControl.arrProfileParameter[7,1].bEnFdbUp			:= FALSE;	
PlantControl.arrProfileParameter[7,1].bEnFdbDown		:= FALSE;	
                          
PlantControl.arrProfileParameter[7,2].bValue			:= FALSE;		
PlantControl.arrProfileParameter[7,2].nValue			:= 0;		
PlantControl.arrProfileParameter[7,2].fValue			:= 0;		
PlantControl.arrProfileParameter[7,2].fDelayUp			:= 0;	
PlantControl.arrProfileParameter[7,2].fDelayDown		:= 0;	
PlantControl.arrProfileParameter[7,2].bEnFdbUp			:= FALSE;	
PlantControl.arrProfileParameter[7,2].bEnFdbDown		:= FALSE;	
                          
PlantControl.arrProfileParameter[7,3].bValue			:= TRUE;		
PlantControl.arrProfileParameter[7,3].nValue			:= 0;		
PlantControl.arrProfileParameter[7,3].fValue			:= 0;		
PlantControl.arrProfileParameter[7,3].fDelayUp			:= 0;	
PlantControl.arrProfileParameter[7,3].fDelayDown		:= 0;	
PlantControl.arrProfileParameter[7,3].bEnFdbUp			:= TRUE;	
PlantControl.arrProfileParameter[7,3].bEnFdbDown		:= FALSE;	
                          
PlantControl.arrProfileParameter[7,4].bValue			:= FALSE;		
PlantControl.arrProfileParameter[7,4].nValue			:= E_BA_Mdlt.eMax;		
PlantControl.arrProfileParameter[7,4].fValue			:= 0;		
PlantControl.arrProfileParameter[7,4].fDelayUp			:= 0;	
PlantControl.arrProfileParameter[7,4].fDelayDown		:= 0;	
PlantControl.arrProfileParameter[7,4].bEnFdbUp			:= FALSE;	
PlantControl.arrProfileParameter[7,4].bEnFdbDown		:= FALSE;	
                          
PlantControl.arrProfileParameter[7,5].bValue			:= TRUE;		
PlantControl.arrProfileParameter[7,5].nValue			:= 0;		
PlantControl.arrProfileParameter[7,5].fValue			:= 0;		
PlantControl.arrProfileParameter[7,5].fDelayUp			:= 0;	
PlantControl.arrProfileParameter[7,5].fDelayDown		:= 0;	
PlantControl.arrProfileParameter[7,5].bEnFdbUp			:= TRUE;	
PlantControl.arrProfileParameter[7,5].bEnFdbDown		:= FALSE;	
                          
PlantControl.arrProfileParameter[7,6].bValue			:= FALSE;		
PlantControl.arrProfileParameter[7,6].nValue			:= E_BA_Mdlt.eMax;		
PlantControl.arrProfileParameter[7,6].fValue			:= 0;		
PlantControl.arrProfileParameter[7,6].fDelayUp			:= 0;	
PlantControl.arrProfileParameter[7,6].fDelayDown		:= 0;	
PlantControl.arrProfileParameter[7,6].bEnFdbUp			:= FALSE;	
PlantControl.arrProfileParameter[7,6].bEnFdbDown		:= FALSE;	
                          
PlantControl.arrProfileParameter[7,7].bValue			:= FALSE;		
PlantControl.arrProfileParameter[7,7].nValue			:= 0;		
PlantControl.arrProfileParameter[7,7].fValue			:= 0;		
PlantControl.arrProfileParameter[7,7].fDelayUp			:= 0;	
PlantControl.arrProfileParameter[7,7].fDelayDown		:= 0;	
PlantControl.arrProfileParameter[7,7].bEnFdbUp			:= FALSE;	
PlantControl.arrProfileParameter[7,7].bEnFdbDown		:= FALSE;	
                          
PlantControl.arrProfileParameter[7,8].bValue			:= FALSE;		
PlantControl.arrProfileParameter[7,8].nValue			:= E_BA_Mdlt.eOff;		
PlantControl.arrProfileParameter[7,8].fValue			:= 0;		
PlantControl.arrProfileParameter[7,8].fDelayUp			:= 0;	
PlantControl.arrProfileParameter[7,8].fDelayDown		:= 0;	
PlantControl.arrProfileParameter[7,8].bEnFdbUp			:= FALSE;	
PlantControl.arrProfileParameter[7,8].bEnFdbDown		:= FALSE;
END_METHOD

METHOD ProfileParameter08
VAR
END_VAR
// Profile LifeSaftyOff
// PlantControl.arrProfileParameter[Profile,Step]
// Step 1 = Erc, 
// Step 2 = PreHtr
// Step 3 = DamperOuA
// Step 4 = FanSupplyAir
// Step 5 = DamperExhA
// Step 6 = FanExtractAir
// Step 7 = Cooler
// Step 8 = EnablingTemperatureControl

PlantControl.arrProfileParameter[8,1].bValue			:= FALSE;		
PlantControl.arrProfileParameter[8,1].nValue			:= 0;
PlantControl.arrProfileParameter[8,1].fValue			:= 0;		
PlantControl.arrProfileParameter[8,1].fDelayUp			:= 0;	
PlantControl.arrProfileParameter[8,1].fDelayDown		:= 0;	
PlantControl.arrProfileParameter[8,1].bEnFdbUp			:= FALSE;	
PlantControl.arrProfileParameter[8,1].bEnFdbDown		:= FALSE;	
                           
PlantControl.arrProfileParameter[8,2].bValue			:= FALSE;		
PlantControl.arrProfileParameter[8,2].nValue			:= 0;		
PlantControl.arrProfileParameter[8,2].fValue			:= 0;		
PlantControl.arrProfileParameter[8,2].fDelayUp			:= 0;	
PlantControl.arrProfileParameter[8,2].fDelayDown		:= 0;	
PlantControl.arrProfileParameter[8,2].bEnFdbUp			:= FALSE;	
PlantControl.arrProfileParameter[8,2].bEnFdbDown		:= FALSE;	
                           
PlantControl.arrProfileParameter[8,3].bValue			:= FALSE;		
PlantControl.arrProfileParameter[8,3].nValue			:= 0;		
PlantControl.arrProfileParameter[8,3].fValue			:= 0;		
PlantControl.arrProfileParameter[8,3].fDelayUp			:= 0;	
PlantControl.arrProfileParameter[8,3].fDelayDown		:= 0;	
PlantControl.arrProfileParameter[8,3].bEnFdbUp			:= FALSE;	
PlantControl.arrProfileParameter[8,3].bEnFdbDown		:= FALSE;	
                           
PlantControl.arrProfileParameter[8,4].bValue			:= FALSE;		
PlantControl.arrProfileParameter[8,4].nValue			:= E_BA_Mdlt.eOff;		
PlantControl.arrProfileParameter[8,4].fValue			:= 0;		
PlantControl.arrProfileParameter[8,4].fDelayUp			:= 0;	
PlantControl.arrProfileParameter[8,4].fDelayDown		:= 0;	
PlantControl.arrProfileParameter[8,4].bEnFdbUp			:= FALSE;	
PlantControl.arrProfileParameter[8,4].bEnFdbDown		:= FALSE;	
                           
PlantControl.arrProfileParameter[8,5].bValue			:= FALSE;		
PlantControl.arrProfileParameter[8,5].nValue			:= 0;		
PlantControl.arrProfileParameter[8,5].fValue			:= 0;		
PlantControl.arrProfileParameter[8,5].fDelayUp			:= 0;	
PlantControl.arrProfileParameter[8,5].fDelayDown		:= 0;	
PlantControl.arrProfileParameter[8,5].bEnFdbUp			:= FALSE;	
PlantControl.arrProfileParameter[8,5].bEnFdbDown		:= FALSE;	
                           
PlantControl.arrProfileParameter[8,6].bValue			:= FALSE;		
PlantControl.arrProfileParameter[8,6].nValue			:= E_BA_Mdlt.eOff;		
PlantControl.arrProfileParameter[8,6].fValue			:= 0;		
PlantControl.arrProfileParameter[8,6].fDelayUp			:= 0;	
PlantControl.arrProfileParameter[8,6].fDelayDown		:= 0;	
PlantControl.arrProfileParameter[8,6].bEnFdbUp			:= FALSE;	
PlantControl.arrProfileParameter[8,6].bEnFdbDown		:= FALSE;	
                           
PlantControl.arrProfileParameter[8,7].bValue			:= FALSE;		
PlantControl.arrProfileParameter[8,7].nValue			:= 0;		
PlantControl.arrProfileParameter[8,7].fValue			:= 0;		
PlantControl.arrProfileParameter[8,7].fDelayUp			:= 0;	
PlantControl.arrProfileParameter[8,7].fDelayDown		:= 0;	
PlantControl.arrProfileParameter[8,7].bEnFdbUp			:= FALSE;	
PlantControl.arrProfileParameter[8,7].bEnFdbDown		:= FALSE;	
                           
PlantControl.arrProfileParameter[8,8].bValue			:= FALSE;		
PlantControl.arrProfileParameter[8,8].nValue			:= E_BA_Mdlt.eOff;		
PlantControl.arrProfileParameter[8,8].fValue			:= 0;		
PlantControl.arrProfileParameter[8,8].fDelayUp			:= 0;	
PlantControl.arrProfileParameter[8,8].fDelayDown		:= 0;	
PlantControl.arrProfileParameter[8,8].bEnFdbUp			:= FALSE;	
PlantControl.arrProfileParameter[8,8].bEnFdbDown		:= FALSE;
END_METHOD

METHOD StepDescription : BOOL
PlantControl.arrStepDescription[1]	:= txtEvent_EnergyRecovery;
PlantControl.arrStepDescription[2]	:= txtEvent_PreRinse;
PlantControl.arrStepDescription[3]	:= txtEvent_DamperOutsideAir;
PlantControl.arrStepDescription[4]	:= txtEvent_SupplyAirFan;
PlantControl.arrStepDescription[5]	:= txtEvent_DamperExhaustAir;
PlantControl.arrStepDescription[6]	:= txtEvent_ExtractAirFan;
PlantControl.arrStepDescription[7]	:= txtEvent_Cooler;
PlantControl.arrStepDescription[8]	:= txtEvent_EnableTemperatureControl;
END_METHOD

END_FUNCTION_BLOCK

(* stored: Version 1.1.0.1, ProductVersion 3.1.4024.15
   POU FB_BA_AC_PlantCmd_AHU_1st_10: Id {48ac3ade-e3bf-4d4a-816c-d36a6b01b44d}, SpecialFunc None
   Folder Profiles: Id {329b977c-5e78-4d3f-8299-11b19a7ebd2c}
   Method CallInit: Id {8ac02f3c-8ce1-4d0a-b131-c512b5b80f0d}
   Method FB_init: Id {0b1f1d12-15bc-4e77-ad63-f5519ca79f66}
   Method ProfileDescription: Id {7e79b98b-68f8-4c90-acdd-4360cb2c75ae}
   Method ProfileParameter01: Id {6ecb2880-09a3-4e75-88cb-6f95e7b3ab01}
   Method ProfileParameter02: Id {eb6fe2a8-1818-4b53-9540-90cfd6b98dbe}
   Method ProfileParameter03: Id {1aabf739-49cd-4e84-89b0-34b45f7e0495}
   Method ProfileParameter04: Id {9b07286a-b0eb-45ad-bdf5-65830f7ff919}
   Method ProfileParameter05: Id {f138942b-5774-4410-89c3-6a51e14fbef3}
   Method ProfileParameter06: Id {e62542bb-8551-440c-8441-14c42ef5deae}
   Method ProfileParameter07: Id {b90d8ab8-4de6-45e7-96d0-82cb5f29bca2}
   Method ProfileParameter08: Id {378e8457-3c50-4807-8fa3-9dd529ab4dca}
   Method StepDescription: Id {7c8449a7-2f63-4af4-9793-cf0e63ee8454} *)
